(* CoDeSys 2.3.9.37 project: Cap12_10_Res.pro *)
(* Libraries: Util.lib 18.5.10 16:14:28, Standard.lib 4.10.05 12:14:46, IecSfc.lib 13.4.06 16:51:28 *)

(* Global variable list: Global_Variables *)
VAR_GLOBAL
   (* Entradas PLC *)
   IW1_Posicion : WORD;   (* Posición real de la valvula *)
   IX2_Error : BOOL;         (* Error en la Válvula *)
    IW2_Caudal : WORD;  (*Lectura del caudalímetro *)
   IX3_Boton : BOOL;    (* puesta en marcha del proceso secuancial *)


   (*Salidas *)
   QW1_SPPosicion : WORD;  (* Consigna de posición para la válvula *)


(*-----------------------------------------------------------------------------------*)

(* Otras variables para la simulación *)
   QX3_ValvulaONOFF: BOOL; (* Orden Abre/Cierra Valvula ON/OFF *)

    (* Variables reales para entradas y salidas *)
    Posicion : REAL;   (*IW1_Posicion  en REAL *)
    Caudal : REAL;   (*IW2_Posicion  en REAL *)
    SPPosicion: REAL; (* QW1_SPPosicion en REAL *)

    (* Variables para el control de la visualización *)
   (* Valvula 1 *)
   Man : BOOL;  (* Manual/Automarico *)
   ManGRAFCET: BOOL;
   RefManual : REAL;  (* SP Manual en lazo abierto*)

   (* PI de la valvula 1 *)
   PropPI : BOOL;
   ManPI : BOOL;  (* Manual/Automatico PI *)
   ManPIGRAFCET: BOOL;
   ManPI_Ent: REAL;  (* Valor de entrada del PI Manual *)
   ManPI_EntGRAFCET: REAL;
   KpPI : REAL := 0.2; (*Parametro Kp del PI *)
   TNPI:REAL := 400;  (* Tiempo Integral del PI *)
  SPPI:REAL := 30;  (* Set Point del PI en modo lazo cerrado *)
  SPPIGRAFCET: REAL;

END_VAR

(* POU PLC_PRG, ST *)
PROGRAM PLC_PRG
VAR
END_VAR
 Proceso();
  EscaladoSenales();
 ProgramaControl();
 Secuencial();
END_PROGRAM

(* POU Proceso, ST *)
PROGRAM Proceso
VAR
       (* Parámetros del sistema posición válvula *)
       K: REAL :=1;
       tau : REAL:=500;
       (* Parámetros del sistema Posición-Caudal *)
       K1: REAL :=0.6;
       tau1 : REAL:=3000;
      (* Variables de tiempo *)
	tact: TIME;
	tactw: DWORD;
	tinc: REAL;
	toldw: DWORD;
      (* Variables del Proceso *)
      Pos : REAL;
     SP_Pos:REAL;
     Caudal:REAL;
      Ciclo1:BOOL:=TRUE;
	EscalaSalida: Escalado;
	IW1R: REAL;
      IW2R:REAL;
	EscalaEntrada: Escalado;
	QW1R: REAL;
	EscalaPos: Escalado;
	EscalaCaudal: Escalado;
END_VAR
  (* Lectura de la consigna de la posición y paso a real *)
  QW1R:=WORD_TO_REAL(QW1_SPPosicion);
  EscalaEntrada(Valor_Ent:=QW1R,Min_Ent:=0,Max_Ent:=4095,Min_Sal:=0,Max_Sal:=100,Valor_Sal=>SP_Pos);

    (* Programa que simula un sistema de primer orden *)
    tact:=TIME();
    tactw:=TIME_TO_DWORD(tact);
    (* Calcula el intervalo de tiempo desde el último ciclo en milisegundos *)
    tinc:=DWORD_TO_REAL(tactw-toldw);
    (* Almacena el valor actual para al próximo ciclo *)
    toldw:=tactw;



    IF Ciclo1=FALSE THEN
        Pos:=Pos+tinc*(K*SP_Pos-Pos)/tau;
        Caudal:=Caudal+tinc*(K1*Pos-Caudal)/tau1;
    ELSE
        Ciclo1:=FALSE;
    END_IF

    EscalaPos(Valor_Ent:=Pos,Min_Ent:=0,Max_Ent:=100,Min_Sal:=0,Max_Sal:=4095,Valor_Sal=>IW1R);
    IW1_Posicion:=REAL_TO_WORD(IW1R);
     EscalaCaudal(Valor_Ent:=Caudal,Min_Ent:=0,Max_Ent:=100,Min_Sal:=0,Max_Sal:=4095,Valor_Sal=>IW2R);
    IW2_Caudal:=REAL_TO_WORD(IW2R);
END_PROGRAM

(* POU Escalado, ST *)
FUNCTION_BLOCK Escalado
VAR_INPUT
	Valor_Ent : REAL;    (* Valor a convertir *)
	Min_Ent : REAL;      (* Valor mínimo de la entrada *)
	Max_Ent : REAL;	  (* Valor máximo de la entrada *)
	Min_Sal : REAL;      (* Valor mínimo de la salida *)
	Max_Sal : REAL;	   (* . Valor máximo de la salida. *)
       ValError : REAL:=-1;    (*Valor al que poner la salida en caso de error *)
END_VAR
VAR_OUTPUT
	Valor_Sal : REAL;   (*. Valor convertido *)
	Error :  BOOL;         (* Se activa cuando el valor de entrada queda fuera de límites *)
END_VAR
VAR
	pendiente: REAL;
END_VAR
Error:= (Valor_Ent>Max_Ent) OR (Valor_Ent<Min_Ent);

IF NOT Error THEN
   pendiente:=(Max_Sal-Min_Sal)/(Max_Ent-Min_Ent);
   Valor_Sal:=Valor_Ent*pendiente+Min_Sal;
ELSE
   Valor_Sal:=ValError;
END_IF
END_FUNCTION_BLOCK

(* POU EscaladoSenales, FBD *)
PROGRAM EscaladoSenales
VAR
	EscalaPos: Escalado;
	EscalaSP: Escalado;
END_VAR
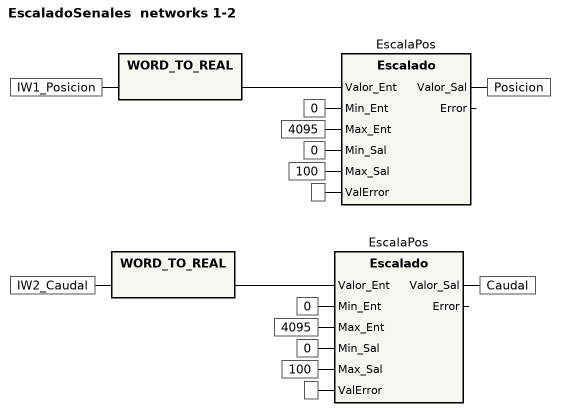
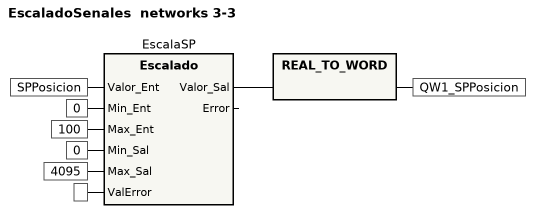
_FBD_ (* Function Block Diagram *)
NETWORK 1
	EscalaPos:Escalado(Valor_Ent: WORD_TO_REAL(IW1_Posicion), Min_Ent: 0, Max_Ent: 4095, Min_Sal: 0, Max_Sal: 100, ValError: ) => Posicion
NETWORK 2
	EscalaPos:Escalado(Valor_Ent: WORD_TO_REAL(IW2_Caudal), Min_Ent: 0, Max_Ent: 4095, Min_Sal: 0, Max_Sal: 100, ValError: ) => Caudal
NETWORK 3
	REAL_TO_WORD(EscalaSP:Escalado(Valor_Ent: SPPosicion, Min_Ent: 0, Max_Ent: 100, Min_Sal: 0, Max_Sal: 4095, ValError: )) => QW1_SPPosicion
_END_FBD_
END_PROGRAM

(* POU ProgramaControl, FBD *)
PROGRAM ProgramaControl
VAR
	Valvula1: ControlValvula;
      PICaudal: ControladorPI;
      PI1Caudal:PIDobleControl;
	Diferencia: REAL;
	LuzValvula: BOOL;
END_VAR
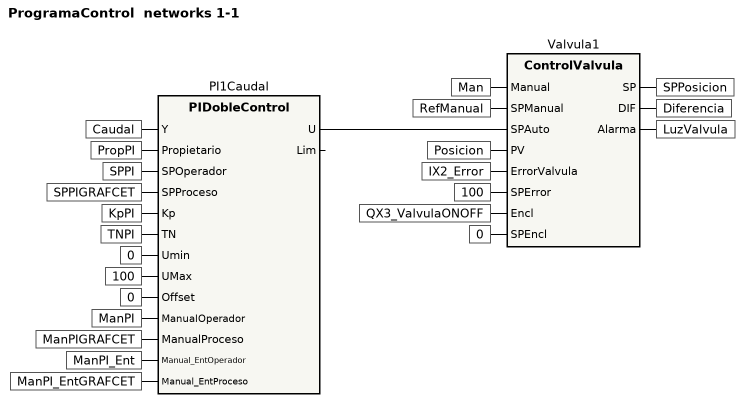
_FBD_ (* Function Block Diagram *)
NETWORK 1
	Valvula1:ControlValvula(Manual: Man, SPManual: RefManual, SPAuto: PI1Caudal:PIDobleControl(Y: Caudal, Propietario: PropPI, SPOperador: SPPI, SPProceso: SPPIGRAFCET, Kp: KpPI, TN: TNPI, Umin: 0, UMax: 100, Offset: 0, ManualOperador: ManPI, ManualProceso: ManPIGRAFCET, Manual_EntOperador: ManPI_Ent, Manual_EntProceso: ManPI_EntGRAFCET), PV: Posicion, ErrorValvula: IX2_Error, SPError: 100, Encl: QX3_ValvulaONOFF, SPEncl: 0, DIF => Diferencia, Alarma => LuzValvula) => SPPosicion
_END_FBD_
(* the same logic as Structured Text *)
(* Network 1 *)
PI1Caudal(Y := Caudal, Propietario := PropPI, SPOperador := SPPI, SPProceso := SPPIGRAFCET, Kp := KpPI, TN := TNPI, Umin := 0, UMax := 100, Offset := 0, ManualOperador := ManPI, ManualProceso := ManPIGRAFCET, Manual_EntOperador := ManPI_Ent, Manual_EntProceso := ManPI_EntGRAFCET);
Valvula1(Manual := Man, SPManual := RefManual, SPAuto := PI1Caudal.U, PV := Posicion, ErrorValvula := IX2_Error, SPError := 100, Encl := QX3_ValvulaONOFF, SPEncl := 0);
Diferencia := Valvula1.DIF;
LuzValvula := Valvula1.Alarma;
SPPosicion := Valvula1.SP;
END_PROGRAM

(* POU ControlValvula, ST *)
FUNCTION_BLOCK ControlValvula
VAR_INPUT
    Manual : BOOL;
    SPManual : REAL;
    SPAuto : REAL;
    PV : REAL;
    ErrorValvula : BOOL;
    SPError : REAL;
     Encl : BOOL;
     SPEncl : REAL;
END_VAR
VAR_OUTPUT
      SP:REAL;
      DIF : REAL;
      Alarma : BOOL;
END_VAR
VAR
	TempoError: TON;
	INTempo: BOOL;
END_VAR
IF MANUAL THEN
     SP:=SPManual;
ELSE
     SP:= SPAuto;
END_IF

(* Se le da prioridad al enclavamiento *)
IF Encl THEN SP:=SPEncl;  END_IF

DIF:=SP-PV;
INTempo:= ABS(DIF)>0.3;
TempoError(IN:=INTempo, PT:=T#10h);

Alarma:=ErrorValvula OR TempoError.Q;
(* Prioridad máxima a la salida de error *)
IF (Alarma) THEN  SP:=SPError;   END_IF
END_FUNCTION_BLOCK

(* POU ControladorPI, ST *)
FUNCTION_BLOCK ControladorPI
VAR_INPUT
	Y :REAL;       (* Variable a controlar. *)
	SP : REAL;    (* Set Point, valor deseado de la variable a controlar.*)
	Kp : REAL := 1;     (* Parámetro del controlador. Proporcionar un valor por defecto de 1.0.*)
       TN : REAL:=1;       (* Parámetro del controlador *)
	Umin  : REAL :=0;   (* Valor mínimo de la salida. Por defecto tendrá el valor 0 *)
	UMax : REAL:=100;   (* Valor máximo de la salida. Por defecto, tendrá un valor 100.0.*)
	Offset :REAL:=0;     (* Cantidad a sumar a la señal del controlador. Por defecto tendrá un valor 0.*)
	Manual : BOOL;      (* TRUE modo manual, FALSE modo automático*)
	Manual_Ent : REAL;   (*Valor para la salida según ecuación (1.3) en modo manual *)
END_VAR
VAR_OUTPUT
	U : REAL;    (*Salida del controlador. *)
      Lim : BOOL;  (*Estará a TRUE si se superan los límites Umin o Umax en la salida *)
END_VAR
VAR
	tact: TIME;
	tactw: DWORD;
	tinc: REAL;
	toldw: DWORD;
	error: REAL;
	ierror: REAL;
      Ciclo1:BOOL :=TRUE;
END_VAR
   (* Calcula el instante de tiempo actual y se pasa a DWORD en milisegundos *)
    tact:=TIME();
    tactw:=TIME_TO_DWORD(tact);
    (* Calcula el intervalo de tiempo desde el último ciclo en milisegundos *)
    tinc:=DWORD_TO_REAL(tactw-toldw);
    (* Almacena el valor actual para al próximo ciclo *)
    toldw:=tactw;

IF Manual THEN
   U:=Manual_Ent+Offset;
   ierror:=0;
ELSE

    (* Calculo error ¨*)
   error:=SP-Y;
   (* Calculo de la integral del error  usando el método de Euler*)
   IF NOT Ciclo1 THEN
       ierror:=ierror+tinc*error;
  END_IF

   (* Calculo de la salida del conttrolador *)
  U:=Kp*(error+(1/TN)*ierror)+Offset;


END_IF


IF Ciclo1 THEN
   U:=Offset;
   Ciclo1:=FALSE;
END_IF


IF U>Umax THEN
     U:=Umax;
ELSE
   IF U<Umin THEN
       U:=Umin;
   END_IF
END_IF

LIM:=(U>Umax) OR  (U<Umin);
END_FUNCTION_BLOCK

(* POU PIDobleControl, FBD *)
FUNCTION_BLOCK PIDobleControl
VAR_INPUT
	Y :REAL;       (* Variable a controlar. *)
       Propietario : BOOL;
	SPOperador : REAL;    (* Set Point, valor deseado de la variable a controlar.*)
       SPProceso : REAL;
	Kp : REAL := 1;     (* Parámetro del controlador. Proporcionar un valor por defecto de 1.0.*)
       TN : REAL:=1;       (* Parámetro del controlador *)
	Umin  : REAL :=0;   (* Valor mínimo de la salida. Por defecto tendrá el valor 0 *)
	UMax : REAL:=100;   (* Valor máximo de la salida. Por defecto, tendrá un valor 100.0.*)
	Offset :REAL:=0;     (* Cantidad a sumar a la señal del controlador. Por defecto tendrá un valor 0.*)
	ManualOperador : BOOL;      (* TRUE modo manual, FALSE modo automático*)
       ManualProceso : BOOL;      (* TRUE modo manual, FALSE modo automático*)
	Manual_EntOperador : REAL;   (*Valor para la salida según ecuación (1.3) en modo manual *)
       Manual_EntProceso : REAL;   (*Valor para la salida según ecuación (1.3) en modo manual *)
END_VAR
VAR_OUTPUT
	U : REAL;    (*Salida del controlador. *)
      Lim : BOOL;  (*Estará a TRUE si se superan los límites Umin o Umax en la salida *)
END_VAR
VAR
	MiPi: ControladorPI;
END_VAR
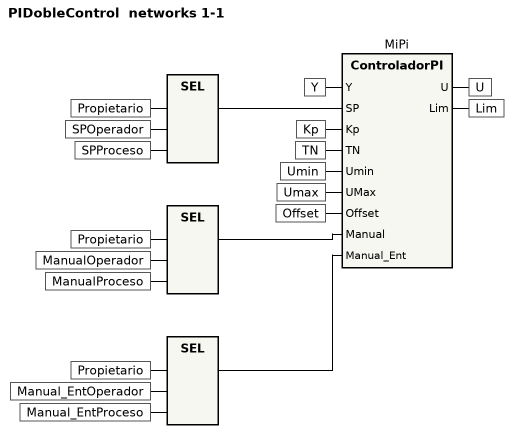
_FBD_ (* Function Block Diagram *)
NETWORK 1
	MiPi:ControladorPI(Y: Y, SP: SEL(Propietario, SPOperador, SPProceso), Kp: Kp, TN: TN, Umin: Umin, UMax: Umax, Offset: Offset, Manual: SEL(Propietario, ManualOperador, ManualProceso), Manual_Ent: SEL(Propietario, Manual_EntOperador, Manual_EntProceso), Lim => Lim) => U
_END_FBD_
(* the same logic as Structured Text *)
(* Network 1 *)
MiPi(Y := Y, SP := SEL(Propietario, SPOperador, SPProceso), Kp := Kp, TN := TN, Umin := Umin, UMax := Umax, Offset := Offset, Manual := SEL(Propietario, ManualOperador, ManualProceso), Manual_Ent := SEL(Propietario, Manual_EntOperador, Manual_EntProceso));
Lim := MiPi.Lim;
U := MiPi.U;
END_FUNCTION_BLOCK

(* POU Secuencial, SFC *)
PROGRAM Secuencial
VAR
	TempoE1: TON;
	TempoE2: TON;
	TempoE3: TON;
END_VAR
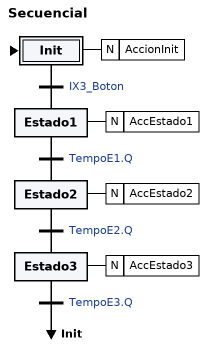
INITIAL_STEP Init:
	AccionInit(N);
END_STEP
TRANSITION FROM Init TO Estado1 := IX3_Boton;
END_TRANSITION
STEP Estado1:
	AccEstado1(N);
END_STEP
TRANSITION FROM Estado1 TO Estado2 := TempoE1.Q;
END_TRANSITION
STEP Estado2:
	AccEstado2(N);
END_STEP
TRANSITION FROM Estado2 TO Estado3 := TempoE2.Q;
END_TRANSITION
STEP Estado3:
	AccEstado3(N);
END_STEP
TRANSITION FROM Estado3 TO Init := TempoE3.Q;
END_TRANSITION
END_PROGRAM
ACTION AccEstado1:
ManPIGRAFCET:=FALSE;
SPPIGRAFCET:=40;
TempoE1(IN:=Estado1.x,PT:=T#30s);
END_ACTION
ACTION AccEstado2:
ManPIGRAFCET:=TRUE;
ManPI_EntGRAFCET:=30;
TempoE2(IN:=Estado2.x,PT:=T#40s);
END_ACTION
ACTION AccEstado3:
ManPIGRAFCET:=FALSE;
SPPIGRAFCET:=10;
TempoE3(IN:=Estado3.x,PT:=T#30s);
END_ACTION
ACTION AccionInit:
ManPIGRAFCET:=TRUE;
ManPI_EntGRAFCET:=0.0;
END_ACTION

(* Visualisation Visu
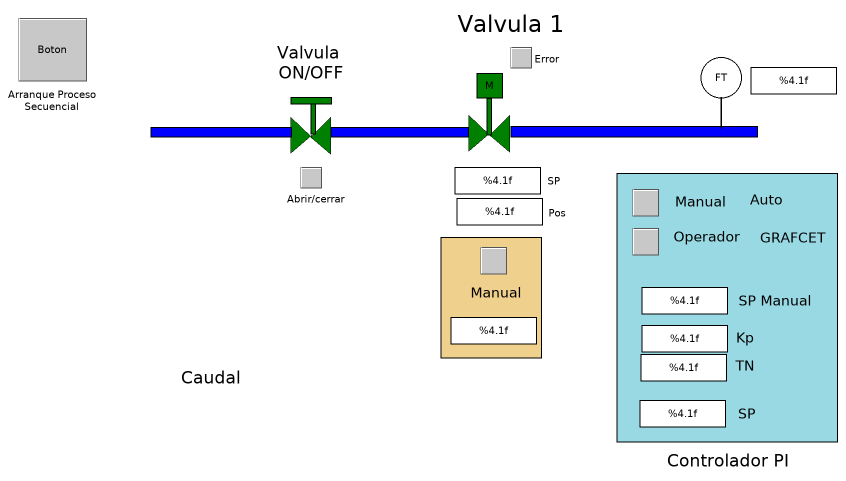
button at (490,260)-(516,287): toggles Man
rectangle at (460,330)-(546,357): text "%4.1f"; shows RefManual; editable 0..100
polygon at (478,128)-(499,164): alarm colour if IX2_Error
polygon at (499,128)-(519,165): alarm colour if IX2_Error
rectangle at (486,86)-(512,111): text "M"; alarm colour if IX2_Error
rectangle at (496,111)-(501,148): alarm colour if IX2_Error
rectangle at (464,180)-(550,207): text "%4.1f"; shows SPPosicion
rectangle at (547,182)-(580,206): text "SP"
rectangle at (550,214)-(583,238): text "Pos"
rectangle at (480,290)-(531,321): text "Manual"
rectangle at (466,211)-(552,238): text "%4.1f"; shows Proceso.Pos
button at (520,60)-(541,81): toggles IX2_Error
rectangle at (540,60)-(573,84): text "Error"
rectangle at (460,20)-(581,54): text "Valvula 1"
polygon at (320,130)-(340,167): alarm colour if QX3_ValvulaONOFF
polygon at (300,130)-(321,166): alarm colour if QX3_ValvulaONOFF
rectangle at (320,110)-(325,147): alarm colour if QX3_ValvulaONOFF
rectangle at (300,110)-(341,117): alarm colour if QX3_ValvulaONOFF
rectangle at (260,50)-(381,101): text "Valvula / ON/OFF"
button at (310,180)-(331,201): toggles QX3_ValvulaONOFF
rectangle at (290,200)-(361,224): text "Abrir/cerrar"
rectangle at (140,370)-(301,411): text "Caudal"
ellipse at (710,70)-(751,111): text "FT"
button at (642,202)-(668,229): toggles ManPI
rectangle at (657,453)-(818,494): text "Controlador PI"
rectangle at (677,199)-(743,230): text "Manual"; alarm colour if ManPI
rectangle at (724,298)-(845,329): text "SP Manual"
rectangle at (651,300)-(737,327): text "%4.1f"; shows ManPI_Ent; editable 0..100
rectangle at (651,338)-(737,365): text "%4.1f"; shows KpPI; editable 0..100
rectangle at (650,367)-(736,394): text "%4.1f"; shows TNPI; editable 0..1000
rectangle at (714,335)-(795,366): text "Kp"
rectangle at (714,363)-(795,394): text "TN"
rectangle at (760,80)-(846,107): text "%4.1f"; shows Proceso.Caudal
rectangle at (649,413)-(735,440): text "%4.1f"; shows SPPI; editable 0..100
rectangle at (716,411)-(797,442): text "SP"
button at (28,31)-(96,94): text "Boton"; taps IX3_Boton
rectangle at (9,83)-(114,144): text "Arranque Proceso / Secuencial"
rectangle at (750,197)-(802,228): text "Auto"; alarm colour if NOT ManPI
button at (642,241)-(668,268): toggles PropPI
rectangle at (681,234)-(752,265): text "Operador"; alarm colour if NOT PropPI
rectangle at (764,235)-(841,266): text "GRAFCET"; alarm colour if PropPI
6 more shapes without text or variables
1 elements of other kinds (tables, trends, ...) not read
*)
